# B&R Automation Studio project databaseTest
Automation Studio 4.9.3.144 SP; technology packages: mapp 5.14.1

## Configuration CP0410

CPU X20CP0410, AutomationRuntime B4.82, Build 4.1.2, Vc V4.72.1

### Task classes (Cpu.sw)
```
Cyclic#4 (cycle 100000 us, tolerance 100000 us):
  dataBaseCo <- Source.dataBaseCom.prg
Libraries: MpDatabase, MpBase, AsHttp, runtime, AsBrStr
```

### Hardware
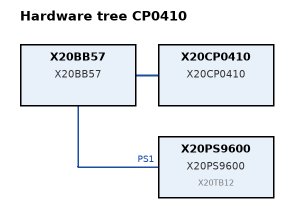
```
X20BB57 : X20BB57 v1.1.1.0
X20CP0410 : X20CP0410 v1.4.0.0  [SL -> X20BB57.SL1]
  Connector IF2:
    ActivateDevice = 1
  ConfigurationID = databaseTest_CP0410
  Simulation = 1
  TimerDeviceType = SWIOTIMER
  Cyclic1Duration = 10000
  Cyclic1Tolerance = 10000
  Cyclic2Duration = 20000
  Cyclic2Tolerance = 20000
  Cyclic3Duration = 50000
  Cyclic3Tolerance = 50000
  Cyclic4Duration = 100000
  Cyclic4Tolerance = 100000
  Cyclic5Duration = 200000
  Cyclic5Tolerance = 200000
  Cyclic6Duration = 500000
  Cyclic6Tolerance = 500000
  Cyclic7Duration = 1000000
  Cyclic7Tolerance = 1000000
  Cyclic8Duration = 10000
  Cyclic8Tolerance = 30000000
X20PS9600 : X20PS9600 v1.3.0.0  [PS -> X20BB57.PS1; SS1 -> X20TB12.SS]
X20TB12 : X20TB12 v1.0.0.0
```

### Config.mpdatabasecore - X20CP0410/mappServices/Config.mpdatabasecore
```
Element gDatabaseCore (Type=mpdatabasecore)
  mapp.Database.Core:
    Name = test
    UserName = plc
    Password = lamisma
    PortNumber = 86
    DBQueries:
      [0]:
        Name = createTable
        Type = CREATE
          TableName = ProductionData
          Columns:
            PV = ::gDbStruct
      [1]:
        Name = insertToProductionData
        Type = INSERT
          Into = ProductionData
          Columns:
            PV = ::gDbStruct
      [2]:
        Name = selectFromProductionData
        Type:
          Select:
            Columns:
              PV = ::gDbStruct
          From = ProductionData
```

## Configuration CP1584

CPU X20CP1584, AutomationRuntime C4.90, Build 4.1.2, Safety 0.0, Vc V4.72.2

### Task classes (Cpu.sw)
```
Libraries: MpDatabase, MpBase, AsHttp, runtime
```

### Hardware
```
X20CP1584 : X20CP1584 v1.8.1.0
```

## Logical view

Binary libraries used (declarations not repeated): operator, runtime, astime, AsIecCon, AsHttp, AsBrStr, MpDatabase 5.12.1, MpBase

### Global.typ - Global data types
```iecst
TYPE
	ProductionData_Db_table_type : 	STRUCT
		id : INT;
		name : STRING[80];
		date : DATE_AND_TIME;
		weight : REAL;
	END_STRUCT;
END_TYPE
```

### Global.var - Global variables
```iecst
VAR
	gDbStruct : ARRAY[0..9] OF ProductionData_Db_table_type;
END_VAR
```

### Package Logical/Libraries - Global libraries

### DataBaseCom.typ - Local data types
```iecst
TYPE
	Db_ctrl_type : 	STRUCT
		cmd : Db_cmd_type;
		param : Db_param_type;
		status : Db_status_type;
		state : Db_state_enum;
	END_STRUCT;
	Db_cmd_type : 	STRUCT
		connectDb : BOOL;
		cancel : BOOL;
		refreshData : BOOL;
		excecuteQuery : BOOL;
		resetError : BOOL;
	END_STRUCT;
	Db_param_type : 	STRUCT
		table : STRING[20];
		queryType : STRING[10];
		dataStructure : REFERENCE TO ProductionData_Db_table_type;
	END_STRUCT;
	Db_status_type : 	STRUCT
		executingQuery : BOOL;
		queryDone : BOOL;
		errorActive : BOOL;
		connectionCounter : USINT;
		dbConnectionActive : BOOL;
		errorState : Db_states_enum;
	END_STRUCT;
	Db_state_enum :Db_states_enum;
	Db_states_enum :
		(
		DB_NO_ERROR := 0,
		DB_DISCONNECTED := 10,
		DB_TRY_CONNECTION := 20,
		DB_WAIT_COMMAND := 30,
		DB_EXECUTE_QUERY := 40,
		DB_ERROR_ACTIVE := 100,
		DB_ERROR_RESET := 101,
		DB_DISABLE_FB := 102
		);
END_TYPE
```

### DataBaseCom.var - Local variables
```iecst
(*Variable principal de control de conexión con base de datos*)
VAR
	gDbCtrl : Db_ctrl_type;
END_VAR
(*BLOQUES DE FUNCIÓN PARA ESTABLECER CONEXIÓN CON DB SQL Y EJECUTAR CONSULTAS*)
VAR
	MpDatabaseCore_SQL : MpDatabaseCore;
	MpDatabase_SQL_Query : MpDatabaseQuery;
END_VAR
(*Variables auxiliares*)
VAR
	queryStr : STRING[80] := ''; (*Variable auxiliar para generar un query*)
END_VAR
(*Constantes del sistema*)
VAR CONSTANT
	CONNECT_TRY_LIMIT : USINT := 3;
	QUERY_SELECT : STRING[10] := 'selectFrom';
	QUERY_INSERT : STRING[10] := 'insertTo';
	QUERY_UPDATE : STRING[10] := 'updateTo';
END_VAR
```

### Program Logical/Source/dataBaseCom (IEC)

#### Main.st - Init, cyclic, exit code
```iecst
(*************************************************************************************

	Este programa genera una interfaz de conexión con una base de datos Microsoft
	SQL (probado con MSSQL Server 2016). Se utiliza el componente de mapp Database
	para facilitar la implementación de la conexión con la base de datos.
	Como middleware, se utiliza un servidor HTTP que se levanta mediante un script
	de Python (probado con Python 3.8.2, ver archivo mappdatabaseconnector3_5_12.py).
	El servidor HTTP es el que se encarga de enviar los queries configurados en el
	componente de mapp Database.

	La conexión con la base de datos es utilizada para almacenar y extraer datos de
	producción mediante un comando de ejecución de query y definiendo cual tabla se
	quiere consultar.

	Versiones utilizadas:

	Mapp Services 5.12

	Microsoft SQL Server 2016

	Python 3.8.2

	MySQL connector v8.0 32-bit (https://dev.mysql.com/downloads/connector/python/)

	MS SQL pyodbc connector v4.0 32- bit (instalado mediante el pip de Python ó se
	puede descargar de:
	https://docs.microsoft.com/en-us/sql/connect/python/python-driver-for-sql-server?view=sql-server-ver15&viewFallbackFrom=sql-server-2017

 *************************************************************************************)

PROGRAM _INIT
	(* Estructura global que contiene las estructuras de intercambio de datos con la
		base de datos Microsoft SQL  *)
	gDbStruct;
	(* Inicializando la máquina de estados *)
	gDbCtrl.state := DB_DISCONNECTED;
END_PROGRAM

PROGRAM _CYCLIC

	//Enlazando las estructuras de datos para almacenar la información de las consultas
	gDbCtrl.param.dataStructure := ADR(gDbStruct);

	CASE gDbCtrl.state OF

		DB_DISCONNECTED:

			IF gDbCtrl.status.connectionCounter <= CONNECT_TRY_LIMIT THEN
				//Preparando bloque de mapp Database
				MpDatabaseCore_SQL.Enable  := TRUE;
				MpDatabaseCore_SQL.MpLink  := ADR(gDatabaseCore);
				//Transición a estado de conexión
				gDbCtrl.state 					 := DB_TRY_CONNECTION;
				gDbCtrl.status.connectionCounter := gDbCtrl.status.connectionCounter + 1;
			ELSIF gDbCtrl.cmd.connectDb THEN
				//Preparando bloque de mapp Database
				MpDatabaseCore_SQL.Enable  := TRUE;
				MpDatabaseCore_SQL.MpLink  := ADR(gDatabaseCore);
				gDbCtrl.cmd.connectDb			 := FALSE;
				//Transición a estado de conexión
				gDbCtrl.state 					 := DB_TRY_CONNECTION;
				gDbCtrl.status.connectionCounter := gDbCtrl.status.connectionCounter + 1;
			ELSE
				//Cuando los intentos de conexión son más de 3, se reinicia el contador
				gDbCtrl.status.connectionCounter := 0;
			END_IF;

		DB_TRY_CONNECTION:

			//Se envía el comando de conexión con SQL
			MpDatabaseCore_SQL.Connect := TRUE;

			IF MpDatabaseCore_SQL.CommandBusy THEN
				(* ESPERANDO A QUE EL BLOQUE ESTABLEZCA LA CONEXIÓN CON SQL *)
			ELSIF MpDatabaseCore_SQL.CommandDone AND MpDatabaseCore_SQL.Connected THEN
				gDbCtrl.status.dbConnectionActive := TRUE;
				gDbCtrl.status.connectionCounter  := 0; //Reset del contador de intentos de conexión
				gDbCtrl.state 					  := DB_WAIT_COMMAND;
			ELSIF gDbCtrl.cmd.cancel THEN
				MpDatabaseCore_SQL.Enable  		  := FALSE;
				MpDatabaseCore_SQL.Connect 		  := FALSE;
				gDbCtrl.state 			   		  := DB_DISCONNECTED;
			ELSIF MpDatabaseCore_SQL.Error THEN
				gDbCtrl.status.errorActive 		  := TRUE;
				gDbCtrl.status.errorState  		  := gDbCtrl.state;
				//Transición al estado de error activo
				gDbCtrl.state 			   		  := DB_ERROR_ACTIVE;
			END_IF;

		DB_WAIT_COMMAND:

			(* Selección de consulta por ejecutar *)

			IF gDbCtrl.cmd.excecuteQuery THEN
				gDbCtrl.cmd.excecuteQuery  := FALSE;
				BuildQuery; //Construyendo la consulta
				gDbCtrl.state 			   := DB_EXECUTE_QUERY;
			ELSIF gDbCtrl.cmd.refreshData THEN
				gDbCtrl.cmd.refreshData	   := FALSE;
				//El refresh de datos en pantalla equivale al query SELECT
				gDbCtrl.param.queryType    := QUERY_SELECT;
				BuildQuery; //Construyendo la consulta
				gDbCtrl.state 			   := DB_EXECUTE_QUERY;
			END_IF;

		DB_EXECUTE_QUERY:

			//Se ejecuta la consulta
			MpDatabase_SQL_Query.Execute := TRUE;
			MpDatabase_SQL_Query();

			IF MpDatabase_SQL_Query.CommandBusy THEN
				(* ESPERANDO A QUE EL BLOQUE DE CONSULTAS FINALICE SU EJECUCIÓN *)
				gDbCtrl.status.executingQuery := TRUE; // Se le vanta bandera que indica ejecución de consulta en proceso
			ELSIF MpDatabase_SQL_Query.CommandDone THEN
				gDbCtrl.status.executingQuery := FALSE; //Reset de bandera
				gDbCtrl.state 			      := DB_WAIT_COMMAND;
				MpDatabase_SQL_Query.Execute  := FALSE;
			ELSIF gDbCtrl.cmd.cancel THEN
				gDbCtrl.status.executingQuery := FALSE; //Reset de bandera
				//Se deshabilita el bloque para dejarlo disponible para próximas consultas
				MpDatabase_SQL_Query.Enable   := FALSE;
				MpDatabase_SQL_Query.Execute  := FALSE;
				MpDatabase_SQL_Query();
				//Validando que el bloque de consultas esté completamente deshabilitado
				IF NOT MpDatabase_SQL_Query.Active THEN
					//Transición al estado de espera de comandos
					gDbCtrl.state 			  := DB_WAIT_COMMAND;
				END_IF;
			ELSIF MpDatabase_SQL_Query.Error THEN
				gDbCtrl.status.errorActive    := TRUE;
				gDbCtrl.status.errorState     := gDbCtrl.state;
				//Transición al estado de error activo
				gDbCtrl.state 			      := DB_ERROR_ACTIVE;
			END_IF;

		DB_ERROR_ACTIVE:

			//Desactivando comandos
			gDbCtrl.cmd.connectDb     	  	  := FALSE;
			gDbCtrl.cmd.excecuteQuery 	  	  := FALSE;
			gDbCtrl.cmd.refreshData       	  := FALSE;
			//Desactivando banderas
			gDbCtrl.status.queryDone  	  	  := FALSE;
			gDbCtrl.status.executingQuery 	  := FALSE;
			gDbCtrl.status.dbConnectionActive := FALSE;

			MpDatabaseCore_SQL.ErrorReset     := gDbCtrl.cmd.resetError;
			MpDatabase_SQL_Query.ErrorReset   := gDbCtrl.cmd.resetError;
			MpDatabase_SQL_Query();

			IF NOT MpDatabaseCore_SQL.Error AND NOT MpDatabase_SQL_Query.Error THEN
				gDbCtrl.state 			   	  := DB_ERROR_RESET;
			END_IF;

		DB_ERROR_RESET:

			//Validando si la base de datos sigue conectada
			IF NOT MpDatabaseCore_SQL.Connected THEN
				gDbCtrl.cmd.resetError     		:= FALSE;
				gDbCtrl.status.errorActive 		:= FALSE;
				gDbCtrl.status.errorState  		:= DB_NO_ERROR;
				//Transición al estado que deshabilita los bloques para intentar una nueva conexión
				gDbCtrl.state 			   		:= DB_DISABLE_FB;
			ELSE
				gDbCtrl.cmd.resetError     		:= FALSE;
				gDbCtrl.status.errorActive 		:= FALSE;
				gDbCtrl.status.errorState  		:= DB_NO_ERROR;
				//Se libera al bloque de consultas
				MpDatabaseCore_SQL.ErrorReset   := FALSE;
				MpDatabase_SQL_Query.ErrorReset := FALSE;
				MpDatabase_SQL_Query.Enable  	:= FALSE;
				MpDatabase_SQL_Query.Execute 	:= FALSE;
				MpDatabase_SQL_Query();
				//Validando que el bloque de consultas esté completamente deshabilitado
				IF NOT MpDatabase_SQL_Query.Active THEN
					//Transición al estado de espera de comandos
					gDbCtrl.state 			    := DB_WAIT_COMMAND;
				END_IF;
			END_IF;

			IF MpDatabaseCore_SQL.Error AND MpDatabase_SQL_Query.Error THEN
				gDbCtrl.status.errorActive 		:= TRUE;
				gDbCtrl.state 			   		:= DB_ERROR_ACTIVE;
			END_IF;

		DB_DISABLE_FB:

			MpDatabaseCore_SQL.Enable    := FALSE;
			MpDatabaseCore_SQL.Connect   := FALSE;
			MpDatabase_SQL_Query.Enable  := FALSE;
			MpDatabase_SQL_Query.Execute := FALSE;
			MpDatabase_SQL_Query();
			IF NOT MpDatabaseCore_SQL.Active AND NOT MpDatabase_SQL_Query.Active THEN
				//Transición al estado que indica desconexión
				gDbCtrl.state 			     := DB_DISCONNECTED;
			END_IF;

	END_CASE;

	(* Ejecutando el bloque principal de conexión con SQL *)
	MpDatabaseCore_SQL();

END_PROGRAM

PROGRAM _EXIT

	(* Deshabilitando el bloque principal de manejo de comuincación con SQL
		para evitar errores después de transferir cambios al PLC            *)
	MpDatabaseCore_SQL.Enable := FALSE;
	MpDatabaseCore_SQL();

END_PROGRAM
```

#### BuildQuery.st
```iecst
ACTION BuildQuery:

	(* Se arma el string que determina cual será
		 la consula que se ejecutará en la base de datos SQL *)
	brsmemset(ADR(queryStr),0,SIZEOF(queryStr));
	brsstrcat(ADR(queryStr),ADR(gDbCtrl.param.queryType));
	brsstrcat(ADR(queryStr),ADR(gDbCtrl.param.table));

	(* Preparando el bloque de mapp para ejecutar la consulta *)
	MpDatabase_SQL_Query.MpLink := ADR(gDatabaseCore);
	MpDatabase_SQL_Query.Enable := TRUE;
	MpDatabase_SQL_Query.Name   := ADR(queryStr);
	MpDatabase_SQL_Query();

END_ACTION
```

#### Variables.var - not listed in the package file held
```iecst
VAR
	MpDatabaseCore_0 : MpDatabaseCore;
	MpDatabaseQuery_0 : MpDatabaseQuery;
	MpDatabaseQuery_1 : MpDatabaseQuery;
	MpDatabaseQuery_2 : MpDatabaseQuery;
END_VAR
```

- DBInterfaceStateDiagram.drawio (not shown)
